// Mitsubishi GX Works2 project: gitTest   PLC: Q06UDV

PROGRAM MAIN
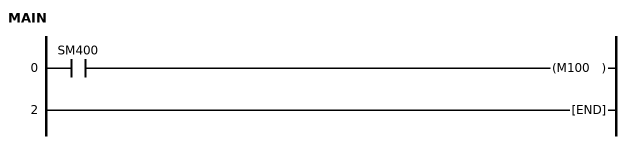
0     LD      SM400
      OUT     M100
2     END
END_PROGRAM

PROGRAM 01  // main0logic
0     END
END_PROGRAM
